% RSLogix 500 project P8_BAK009.RSS, saved by version 12.00.00.00 %
PROJECT "UNTITLED"    % processor: Bul.1763 MicroLogix 1100 Series B %

PROGRAM FILES
  LAD 2 "CNTRL"  4 rungs
  LAD 3 "IO"  3 rungs
  LAD 4 "MAIN"  4 rungs

DATA FILES
  O0 OUTPUT  4 elements
  I1 INPUT  6 elements
  S2 STATUS  66 elements
  B3 BINARY  1 elements
  T4 TIMER  1 elements
  C5 COUNTER  1 elements
  R6 CONTROL  1 elements
  N7 INTEGER  6 elements
  F8 FLOAT  3 elements

LADDER 2 "CNTRL"
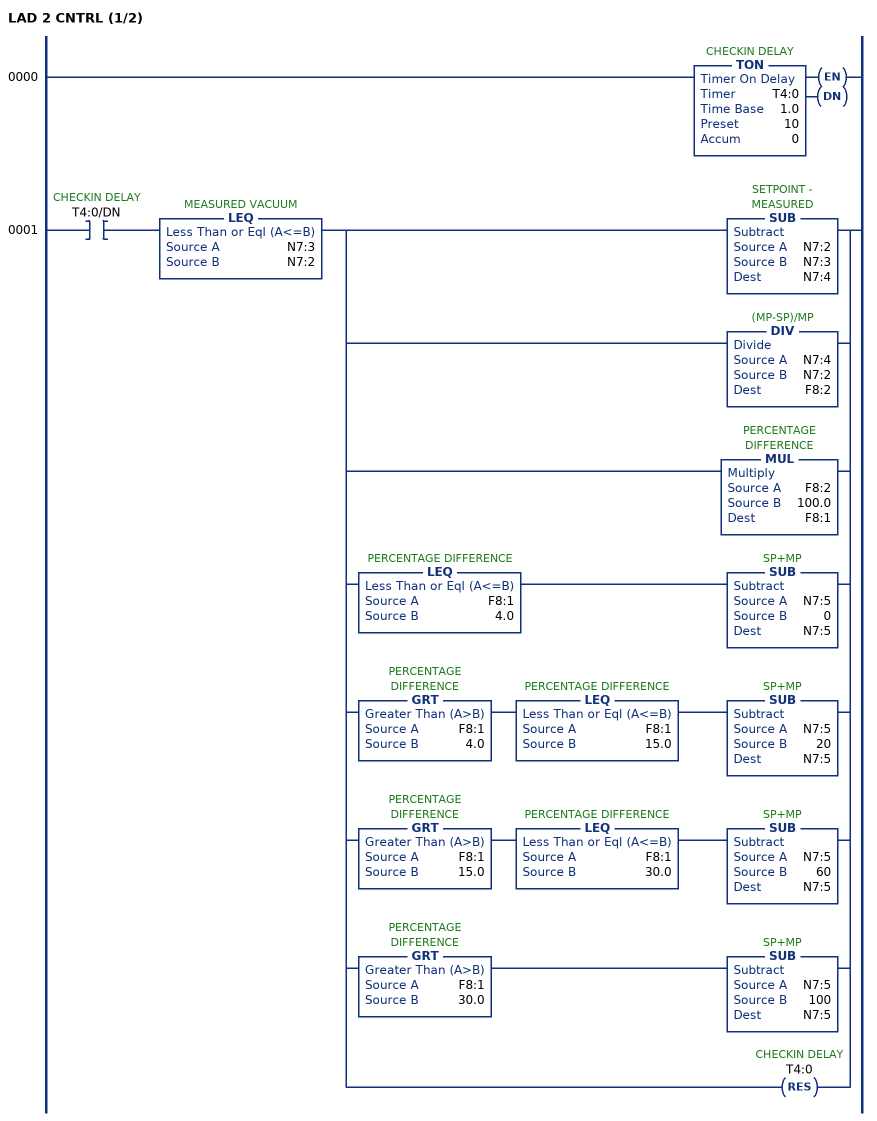
% Rung: 0 %
SOR TON T4:0 1.0 10 0 EOR
%   T4:0  "CHECKIN DELAY" %
% Rung: 1 %
SOR XIC T4:0/DN LEQ N7:3 N7:2 BST SUB N7:2 N7:3 N7:4 NXB DIV N7:4 N7:2 F8:2 NXB MUL F8:2 100.0 F8:1 NXB LEQ F8:1 4.0 SUB N7:5 0 N7:5 NXB GRT F8:1 4.0 LEQ F8:1 15.0 SUB N7:5 20 N7:5 NXB GRT F8:1 15.0 LEQ F8:1 30.0 SUB N7:5 60 N7:5 NXB GRT F8:1 30.0 SUB N7:5 100 N7:5 NXB RES T4:0 BND EOR
%   T4:0  "CHECKIN DELAY" %
%   N7:3  "MEASURED VACUUM" %
%   N7:2  "VACUUM SETPOINT" %
%   N7:4  "SETPOINT - MEASURED" %
%   F8:2  "(MP-SP)/MP" %
%   F8:1  "PERCENTAGE DIFFERENCE" %
%   N7:5  "SP+MP" %

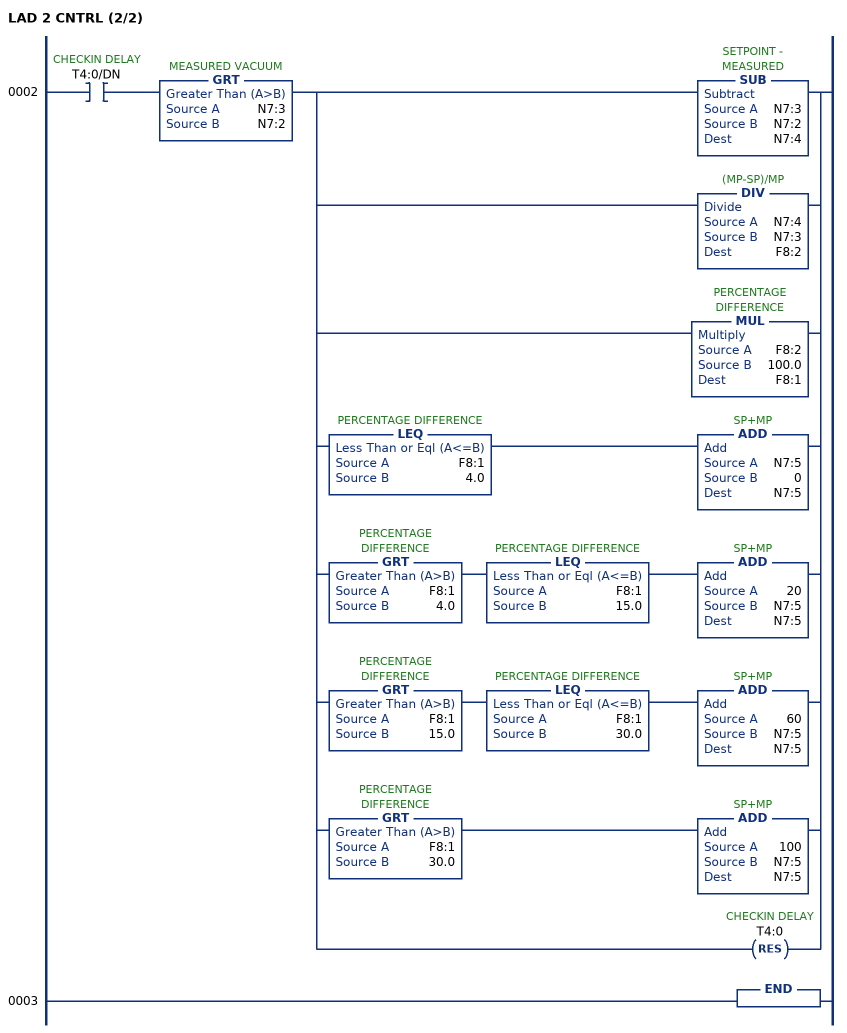
% Rung: 2 %
SOR XIC T4:0/DN GRT N7:3 N7:2 BST SUB N7:3 N7:2 N7:4 NXB DIV N7:4 N7:3 F8:2 NXB MUL F8:2 100.0 F8:1 NXB LEQ F8:1 4.0 ADD N7:5 0 N7:5 NXB GRT F8:1 4.0 LEQ F8:1 15.0 ADD 20 N7:5 N7:5 NXB GRT F8:1 15.0 LEQ F8:1 30.0 ADD 60 N7:5 N7:5 NXB GRT F8:1 30.0 ADD 100 N7:5 N7:5 NXB RES T4:0 BND EOR
%   T4:0  "CHECKIN DELAY" %
%   N7:3  "MEASURED VACUUM" %
%   N7:2  "VACUUM SETPOINT" %
%   N7:4  "SETPOINT - MEASURED" %
%   F8:2  "(MP-SP)/MP" %
%   F8:1  "PERCENTAGE DIFFERENCE" %
%   N7:5  "SP+MP" %
% Rung: 3 %
SOR END EOR

LADDER 3 "IO"
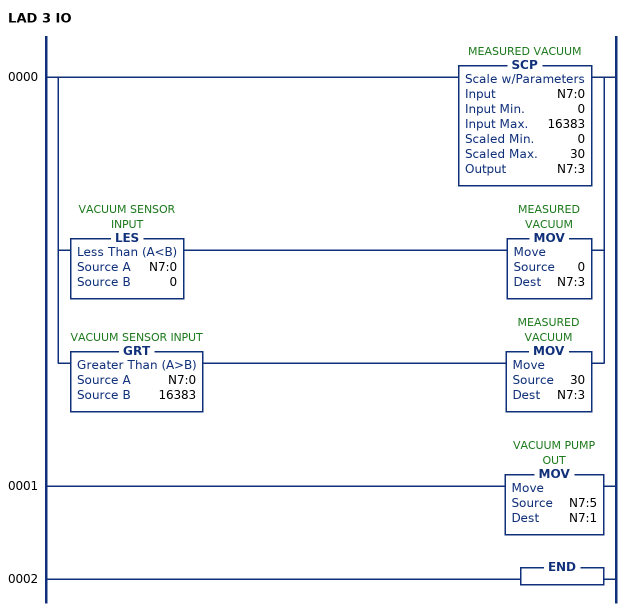
% Rung: 0 %
SOR BST SCP N7:0 0 16383 0 30 N7:3 NXB LES N7:0 0 MOV 0 N7:3 NXB GRT N7:0 16383 MOV 30 N7:3 BND EOR
%   N7:0  "VACUUM SENSOR INPUT" %
%   N7:3  "MEASURED VACUUM" %
% Rung: 1 %
SOR MOV N7:5 N7:1 EOR
%   N7:5  "SP+MP" %
%   N7:1  "VACUUM PUMP OUT" %
% Rung: 2 %
SOR END EOR

LADDER 4 "MAIN"
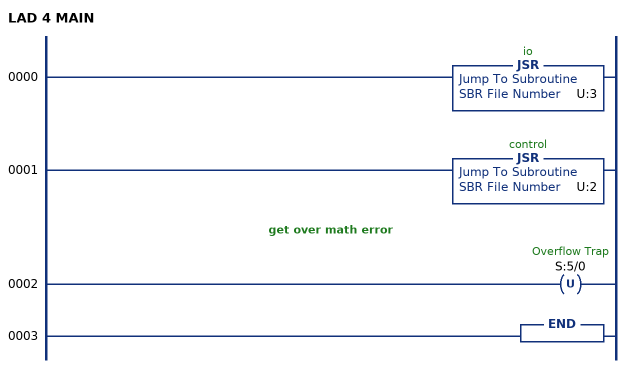
% Rung: 0 %  % edit flag set %
SOR JSR U:3 EOR
%   U:3  "io" %
% Rung: 1 %  % edit flag set %
SOR JSR U:2 EOR
%   U:2  "control" %
% Rung: 2 %  % edit flag set %
% TITLE: get over math error %
SOR OTU S:5/0 EOR
%   S:5/0  "Overflow Trap" %
% Rung: 3 %
SOR END EOR

OTHER DOCUMENTED ADDRESSES
  F8:0  "(SP-MP)/((MP+SP)/2)"

DATA TABLE (non-zero values as saved)
DATA T4
% .PRE .ACC %
% T4:0 % 10 0
DATA F8
% F8:0 % 0.06896552 6.896552 14.5
